{attribute 'GeneratedUsingTerminal: EL3602-0002-0016'}
{attribute addProperty BoxType "EL3602-0002-0016"}
{attribute addProperty Id "AI_Inputs_Channel_1AT %I*AI_Inputs_Channel_4521310411AI_Inputs_Channel_2AT %I*AI_Inputs_Channel_4521310411WcStateAT %I*WcState_9091E0EB2InfoDataAT %I*InfoData_94A18F5E2"}
{attribute addProperty CRC "266334086"}
{attribute addProperty Size "26"}
TYPE EL3602_0FDFEF86 EXTENDS EtcSlaveTerminalBase_947E5A46 :
STRUCT
	{attribute addProperty Name "AI_Inputs_Channel_1"}
	AI_Inputs_Channel_1 : AI_Inputs_Channel_45213104;
	{attribute addProperty Name "AI_Inputs_Channel_2"}
	AI_Inputs_Channel_2 : AI_Inputs_Channel_45213104;
	{attribute addProperty Name "WcState"}
	WcState : WcState_9091E0EB;
	{attribute addProperty Name "InfoData"}
	InfoData : InfoData_94A18F5E;
END_STRUCT
END_TYPE

(* stored: Version 1.2.0.0, ProductVersion 3.1.4024.9
   DUT EL3602_0FDFEF86: Id {2700c1c9-6711-433c-8bd0-b9ecf390e239} *)
